Staubli VAL3: N12_AproAmpolla.pgx

program N12_AproAmpolla()
  local pointRx l_pAproAmpolla
begin

  // Anar a l'aproximació del punt d'agafar líquid de l'ampolla
  l_pAproAmpolla=pAmpolla[aioGet(aiNumAmpolla)]
  l_pAproAmpolla.trsf.x=l_pAproAmpolla.trsf.x+nXOffset
  l_pAproAmpolla.trsf.y=l_pAproAmpolla.trsf.y+nYOffset
  l_pAproAmpolla.trsf.z=l_pAproAmpolla.trsf.z+nZOffset

  if nZApro>0
    l_pAproAmpolla.trsf.z=l_pAproAmpolla.trsf.z+nZApro
  else
    l_pAproAmpolla.trsf.z=l_pAproAmpolla.trsf.z+100
  endIf

  movel(l_pAproAmpolla,tToolActiva,mLent)
  waitEndMove()

  bTaskDone=true
end
